// TIA Portal V20 export
TYPE "HMI_MonDi08"
   STRUCT
      Flut1TmIn : Real;   // Fluttering Time [s]
      Flut2TmIn : Real;   // Fluttering Time [s]
      Flut3TmIn : Real;   // Fluttering Time [s]
      Flut4TmIn : Real;   // Fluttering Time [s]
      Flut5TmIn : Real;   // Fluttering Time [s]
      Flut6TmIn : Real;   // Fluttering Time [s]
      Flut7TmIn : Real;   // Fluttering Time [s]
      Flut8TmIn : Real;   // Fluttering Time [s]
      OnOp : Bool;   // 1=On Mode: On Mode by Operator
      OosOp : Bool;   // 1=Oos Mode: Oos Mode by Operator
      Out1_ST : Byte;
      Out2_ST : Byte;
      Out3_ST : Byte;
      Out4_ST : Byte;
      Out5_ST : Byte;
      Out6_ST : Byte;
      Out7_ST : Byte;
      Out8_ST : Byte;
      OS_PermOut : DWord := DWORD#16#FFFF_FFFF;   // Operator Permission: Output for OS
      OS_PermLog : DWord := DWORD#16#FFFF_FFFF;   // Operator Permission: Output for OS
      OpSt_Out : DWord;   // Enabled operator stations
      ST_Worst : Byte := BYTE#16#80;   // Worst Signal Status
      Status1 : DWord;   // Status1 Word
      Status2 : DWord;   // Status2 Word
      Status3 : DWord;   // Status3 Word
      AlarmState { ExternalWritable := 'False'} : Word;
   END_STRUCT;
END_TYPE
